(* IEC 61131-3 sources: plc-home-automation/home_automation/lighting_heating_updated/src/ventillation, 4 files *)

(* ---- VentillationGlobals.st ---- *)
VAR_GLOBAL CONSTANT

  C_NILAN_READ_COMMAND_GROUP : USINT          := 01;
  C_NILAN_SET_VENTILLATION_LEVEL_COMMAND_GROUP : USINT  := 02;
  C_NILAN_SET_DESIRED_TEMPERATURE_COMMAND_GROUP : USINT := 03;

  C_NUMBER_OF_NILAN_COMMANDS : USINT := 8;

  C_NILAN_STATUS_COMMAND_INDEX : USINT                    := 1;
  C_NILAN_STATUS_COMMAND_SIZE : UINT                        := 17;
  C_NILAN_ACTUAL_OPERATION_INDEX : USINT                  := 2;
  C_NILAN_ACTUAL_OPERATION_COMMAND_SIZE :UINT               := 4;
  C_NILAN_ACTUAL_VENTILLATION_INDEX : USINT               := 3;
  C_NILAN_ACTUAL_VENTILLATION_COMMAND_SIZE : UINT           := 5;
  C_CORE_DIAGNOSTICS_INDEX : USINT                        := 4;
  C_CORE_DIAGNOSTICS_COMMAND_SIZE : UINT                   := 23;
  C_CONTROLLED_TEMPERATURES_INDEX : USINT                 := 5;
  C_CONTROLLED_TEMPERATURES_COMMAND_SIZE : UINT             := 7;
  C_NILAN_SET_VENTILLATION_LEVEL_INDEX : USINT            := 6;
  C_NILAN_SET_VENTILLATION_LEVEL_COMMAND_SIZE : UINT        := 1;
  C_NILAN_SET_DESIRED_TEMPERATURE_INDEX : USINT           := 7;
  C_NILAN_SET_DESIRED_TEMPERATURE_COMMAND_SIZE : UINT       := 1;
  C_NILAN_ACTUAL_DISPLAY_GROUP_01_INDEX : UINT            := 8;
  C_NILAN_ACTUAL_DISPLAY_GROUP_01_COMMAND_SIZE : UINT       := 10;

  C_NILAN_MODBUS_ADDRESS : USINT := 30;

  C_NORMAL_VENTILLATION_LEVEL : INT := 1;
  C_BYPASS_VENTILLATION_LEVEL : INT := 3;

END_VAR

VAR_GLOBAL

  // User control
  PRESENCE_BASED_VENTILLATION_CONTROL   : BOOL := FALSE;
  COOLING_PRIORITY_VENTILLATION_CONTROL : BOOL := FALSE;

  // Read
  NILAN_COMMANDS : ARRAY [1..C_NUMBER_OF_NILAN_COMMANDS] OF TCmdStruct;

  NILAN_COMMAND_SIZES : ARRAY [1..C_NUMBER_OF_NILAN_COMMANDS] OF UINT;
  NILAN_COMMAND_BASE_ADRESSES : ARRAY [1..C_NUMBER_OF_NILAN_COMMANDS] OF UINT;
  NILAN_COMMAND_MODBUS_FNC : ARRAY [1..C_NUMBER_OF_NILAN_COMMANDS] OF USINT;
  NILAN_COMMAND_COMMAND_GROUP : ARRAY [1..C_NUMBER_OF_NILAN_COMMANDS] OF USINT;
  NILAN_COMMAND_DATA : ARRAY [1..C_NUMBER_OF_NILAN_COMMANDS] OF PTR_TO INT;

  NILAN_STATUS : ARRAY                    [1..C_NILAN_STATUS_COMMAND_SIZE] OF INT;
  NILAN_ACTUAL_OPERATION : ARRAY          [1..C_NILAN_ACTUAL_OPERATION_COMMAND_SIZE] OF INT;
  NILAN_ACTUAL_VENTILLATION : ARRAY       [1..C_NILAN_ACTUAL_VENTILLATION_COMMAND_SIZE] OF INT;
  NILAN_CORE_DIAGNOSTICS : ARRAY          [1..C_CORE_DIAGNOSTICS_COMMAND_SIZE] OF INT;
  NILAN_CONTROLLED_TEMPARATURES : ARRAY   [1..C_CONTROLLED_TEMPERATURES_COMMAND_SIZE] OF INT;
  NILAN_ACTUAL_DISPLAY_GROUP_01 : ARRAY   [1..C_NILAN_ACTUAL_DISPLAY_GROUP_01_COMMAND_SIZE] OF INT;

  NILAN_DESIRED_VENTILLATION_LEVEL : INT := 0;
  NILAN_DESIRED_TEMPERATURE        : INT := 24;
  NILAN_DESIRED_TEMPERATURE_SCALED : INT := 2400;

  // Alarms and warninrgs
  NILAN_ACTIVE_ERROR : BOOL := FALSE;
  NILAN_USER_FUNCTION : BOOL := FALSE;
  NILAN_AIR_FILTER_ALARM : BOOL := FALSE;

  // Ventillation
  NILAN_ACTUAL_VENTILLATION_SETPOINT          : INT := 0;
  NILAN_ACTUAL_VENTILLATION_INLET_FAN_LEVEL   : INT := 0;
  NILAN_ACTUAL_VENTILLATION_OUTLET_FAN_LEVEL  : INT := 0;
  NILAN_ACTUAL_VENTILLATION_AVERAGE_FAN_LEVEL : REAL := 0;

  // Core diagnostics (telemetry)
  NILAN_CONTROLLER_BOARD_TEMPERATURE : REAL := 0;

  NILAN_FRESH_AIR_INTAKE_TEMPERATURE    : REAL := 0;
  NILAN_INLET_TEMPERATURE_BEFORE_HEATER : REAL := 0;
  NILAN_ROOM_EXHAUST_TEMPERATURE        : REAL := 0;
  NILAN_OUTLET_TEMPERATURE              : REAL := 0;
  NILAN_CONDENSER_TEMPERATURE           : REAL := 0;
  NILAN_EVAPORATOR_TEMPERATURE          : REAL := 0;
  NILAN_INLET_TEMPERATURE_AFTER_HEATER  : REAL := 0;

  NILAN_OUTDOOR_TEMPERATURE : REAL := 0;

  NILAN_HEATING_SURFACE_TEMPERATURE : INT := 0;
  NILAN_EXTERNAL_ROOM_TEMPERATURE : INT := 0;
  NILAN_HOT_WATER_TOP_TEMPERATURE : INT := 0;
  NILAN_HOT_WATER_BOTTOM_TEMPERATURE : INT := 0;
  NILAN_EK_RETURN_TEMPERATURE : INT := 0;
  NILAN_EK_SUPPLY_TEMPERATURE : INT := 0;
  NILAN_USER_PANEL_ROOM_TEMPERATURE : INT := 0;
  NILAN_AUX_TEMPERATURE_HOTWATER_ANODE : INT := 0;
  NILAN_PREHEATER_OR_EARTH_TUBE_AIR_INTAKE_TEMPERATURE : INT := 0;
  NILAN_PRESSURE_PIBE_TEMPERATURE : INT := 0;
  NILAN_SUCTION_PRESSURE : INT := 0;
  NILAN_DISCHAGE_PRESSURE : INT := 0;
  NILAN_HUMIDITY_SENSOR_VALUE : REAL := 0;
  NILAN_CARBON_DIOXIDE_SENSOR_VALUE : INT := 0;
  NILAN_BYPASS_IS_ENABLED : BOOL := FALSE;

  // Furhter diagnostics
  NILAN_DAYS_SINCE_LAST_FILTER_CHANGE : INT := 0;
  NILAN_ACTUAL_CONTROLLED_TEMPERATURE : REAL := 0;

  NILAN_PASSIVE_HEAT_EXCHANGER_EFFICIENCY : REAL := 0;

END_VAR

(* ---- Ventillation.st ---- *)
PROGRAM VentillationControl

  VAR_INPUT
  END_VAR
  VAR_OUTPUT
  END_VAR
  VAR
     commUnit: fbModbusRTUmas2;
     modbusErrorMessage: String;

     presenceBasedDisable                 : BOOL := FALSE;
     coolingNeeded                        : BOOL := FALSE;

     setPresenceBasedVentillationToZero   : R_TRIG;
     setPresenceBasedVentillationToActive : F_TRIG;

     setCoolingBasedVentillationToZero    : F_TRIG;
     setCoolingBasedVentillationToActive  : R_TRIG;

     activateBypassVentialltionLevel      : R_TRIG;
     deactivateBypassVentialltionLevel    : F_TRIG;

     formerNilanDesiredVentillationLevel : INT := 0;
     formerNilanDesiredTemperature       : INT := 0;
     actualModbusCommandGroup            : USINT := C_NILAN_READ_COMMAND_GROUP;
  END_VAR
  VAR_TEMP
  END_VAR

  NILAN_DESIRED_TEMPERATURE_SCALED := NILAN_DESIRED_TEMPERATURE*100;

  coolingNeeded := (INT_TO_REAL(NILAN_DESIRED_TEMPERATURE) < NILAN_ACTUAL_CONTROLLED_TEMPERATURE) AND COOLING_PRIORITY_VENTILLATION_CONTROL;
  presenceBasedDisable := (GONE_FOR_5_HOURS OR (ALARM_ACTIVE AND GONE_FOR_5_HOURS)) AND NOT coolingNeeded AND PRESENCE_BASED_VENTILLATION_CONTROL;

  setPresenceBasedVentillationToZero(CLK := presenceBasedDisable);
  setPresenceBasedVentillationToACtive(CLK := presenceBasedDisable);

  setCoolingBasedVentillationToZero(CLK := coolingNeeded);
  setCoolingBasedVentillationToActive(CLK := coolingNeeded);

  activateBypassVentialltionLevel(CLK := NILAN_BYPASS_IS_ENABLED);
  deactivateBypassVentialltionLevel(CLK := NILAN_BYPASS_IS_ENABLED);

  // Turn off ventillation when no cooling is required and we're not at home
  IF setPresenceBasedVentillationToZero.Q THEN
    NILAN_DESIRED_VENTILLATION_LEVEL := 0;
  // Turn on ventillation someone is at home or we need cooling
  ELSIF setPresenceBasedVentillationToActive.Q OR setCoolingBasedVentillationToActive.Q THEN
    IF NILAN_BYPASS_IS_ENABLED THEN
      NILAN_DESIRED_VENTILLATION_LEVEL := C_BYPASS_VENTILLATION_LEVEL;
    ELSE
      NILAN_DESIRED_VENTILLATION_LEVEL := C_NORMAL_VENTILLATION_LEVEL;
    END_IF;
  END_IF;

  IF activateBypassVentialltionLevel.Q THEN
    IF NILAN_DESIRED_VENTILLATION_LEVEL < C_BYPASS_VENTILLATION_LEVEL THEN
      NILAN_DESIRED_VENTILLATION_LEVEL := C_BYPASS_VENTILLATION_LEVEL;
    END_IF;
  END_IF;

  IF deactivateBypassVentialltionLevel.Q THEN
    IF NILAN_DESIRED_VENTILLATION_LEVEL > C_NORMAL_VENTILLATION_LEVEL THEN
      NILAN_DESIRED_VENTILLATION_LEVEL := C_NORMAL_VENTILLATION_LEVEL;
    END_IF;
  END_IF;

  IF NOT formerNilanDesiredVentillationLevel = NILAN_DESIRED_VENTILLATION_LEVEL THEN

     actualModbusCommandGroup := C_NILAN_SET_VENTILLATION_LEVEL_COMMAND_GROUP;

     IF commUnit.LastCmd = C_NILAN_SET_VENTILLATION_LEVEL_INDEX THEN
       formerNilanDesiredVentillationLevel := NILAN_DESIRED_VENTILLATION_LEVEL;
     END_IF;

  ELSIF NOT formerNilanDesiredTemperature = NILAN_DESIRED_TEMPERATURE THEN

     actualModbusCommandGroup := C_NILAN_SET_DESIRED_TEMPERATURE_COMMAND_GROUP;

     IF commUnit.LastCmd = C_NILAN_SET_DESIRED_TEMPERATURE_INDEX THEN
       formerNilanDesiredTemperature := NILAN_DESIRED_TEMPERATURE;
     END_IF;

  ELSE

    actualModbusCommandGroup := C_NILAN_READ_COMMAND_GROUP;

  END_IF;

  commUnit(EN := true, GrSel := actualModbusCommandGroup, MaxCmd := C_NUMBER_OF_NILAN_COMMANDS,
             chanCode := CH2_uni, Endian := 0, Commands := NILAN_COMMANDS[1],
             MBtimeOut := T#30s, Delay := T#500ms);

  IF commUnit.ErrCode > 0 THEN
    GetModbusErrTxt(commUnit.ErrCode, modbusErrorMessage);
  END_IF;

  IF commUnit.Done THEN
     actualModbusCommandGroup := C_NILAN_READ_COMMAND_GROUP;
  END_IF;

  // Copy ventillation telemetry to global storage variables
  NILAN_USER_FUNCTION := INT_TO_BOOL(NILAN_STATUS[1]);
  NILAN_AIR_FILTER_ALARM := INT_TO_BOOL(NILAN_STATUS[2]);
  NILAN_ACTUAL_VENTILLATION_SETPOINT          := NILAN_ACTUAL_VENTILLATION[1];
  NILAN_ACTUAL_VENTILLATION_INLET_FAN_LEVEL   := NILAN_ACTUAL_VENTILLATION[2];
  NILAN_ACTUAL_VENTILLATION_OUTLET_FAN_LEVEL  := NILAN_ACTUAL_VENTILLATION[3];
  NILAN_ACTUAL_VENTILLATION_AVERAGE_FAN_LEVEL := INT_TO_REAL(NILAN_ACTUAL_VENTILLATION_INLET_FAN_LEVEL + NILAN_ACTUAL_VENTILLATION_OUTLET_FAN_LEVEL)/2;

  NILAN_CONTROLLER_BOARD_TEMPERATURE := INT_TO_REAL(NILAN_CORE_DIAGNOSTICS[1]) / 100;
  NILAN_FRESH_AIR_INTAKE_TEMPERATURE := INT_TO_REAL(NILAN_CORE_DIAGNOSTICS[2]) / 100;
  NILAN_INLET_TEMPERATURE_BEFORE_HEATER := INT_TO_REAL(NILAN_CORE_DIAGNOSTICS[3]) / 100;
  NILAN_ROOM_EXHAUST_TEMPERATURE := INT_TO_REAL(NILAN_CORE_DIAGNOSTICS[4]) / 100;
  NILAN_OUTLET_TEMPERATURE := INT_TO_REAL(NILAN_CORE_DIAGNOSTICS[5]) / 100;
  NILAN_CONDENSER_TEMPERATURE := INT_TO_REAL(NILAN_CORE_DIAGNOSTICS[6]) / 100;
  NILAN_EVAPORATOR_TEMPERATURE := INT_TO_REAL(NILAN_CORE_DIAGNOSTICS[7]) / 100;
  NILAN_INLET_TEMPERATURE_AFTER_HEATER := INT_TO_REAL(NILAN_CORE_DIAGNOSTICS[8]) / 100;
  NILAN_OUTDOOR_TEMPERATURE := INT_TO_REAL(NILAN_CORE_DIAGNOSTICS[9]) / 100;
  NILAN_HEATING_SURFACE_TEMPERATURE := NILAN_CORE_DIAGNOSTICS[10];
  NILAN_EXTERNAL_ROOM_TEMPERATURE := NILAN_CORE_DIAGNOSTICS[11];
  NILAN_HOT_WATER_TOP_TEMPERATURE := NILAN_CORE_DIAGNOSTICS[12];
  NILAN_HOT_WATER_BOTTOM_TEMPERATURE := NILAN_CORE_DIAGNOSTICS[13];
  NILAN_EK_RETURN_TEMPERATURE := NILAN_CORE_DIAGNOSTICS[14];
  NILAN_EK_SUPPLY_TEMPERATURE := NILAN_CORE_DIAGNOSTICS[15];
  NILAN_USER_PANEL_ROOM_TEMPERATURE := NILAN_CORE_DIAGNOSTICS[16];
  NILAN_AUX_TEMPERATURE_HOTWATER_ANODE := NILAN_CORE_DIAGNOSTICS[17];
  NILAN_PREHEATER_OR_EARTH_TUBE_AIR_INTAKE_TEMPERATURE := NILAN_CORE_DIAGNOSTICS[18];
  NILAN_PRESSURE_PIBE_TEMPERATURE := NILAN_CORE_DIAGNOSTICS[19];
  NILAN_SUCTION_PRESSURE := NILAN_CORE_DIAGNOSTICS[20];
  NILAN_DISCHAGE_PRESSURE := NILAN_CORE_DIAGNOSTICS[21];
  NILAN_HUMIDITY_SENSOR_VALUE := INT_TO_REAL(NILAN_CORE_DIAGNOSTICS[22])/100;
  NILAN_CARBON_DIOXIDE_SENSOR_VALUE := NILAN_CORE_DIAGNOSTICS[23];

  NILAN_DAYS_SINCE_LAST_FILTER_CHANGE := NILAN_ACTUAL_DISPLAY_GROUP_01[7];
  NILAN_BYPASS_IS_ENABLED := INT_TO_BOOL(NILAN_ACTUAL_DISPLAY_GROUP_01[1]);

  NILAN_ACTUAL_CONTROLLED_TEMPERATURE := INT_TO_REAL(NILAN_CONTROLLED_TEMPARATURES[3])/100;

  // This should by scaled by 100 according to the docs, but then I have 100%+ efficiency
  NILAN_PASSIVE_HEAT_EXCHANGER_EFFICIENCY := INT_TO_REAL(NILAN_CONTROLLED_TEMPARATURES[5])/100;

  // Flagging errors requiring physical attention
  NILAN_ACTIVE_ERROR := FALSE;

  IF NILAN_USER_FUNCTION THEN
    NILAN_ACTIVE_ERROR := TRUE;
  END_IF;

END_PROGRAM

(* ---- Ventillation_Control.st ---- *)
TYPE

  TemperatureDataBlock : STRUCT
    controllerBoardTemperature : REAL;
    IntakeTemperature : REAL;
    inletTemperature : REAL;
    exhaustTemparature : REAL;
    outletTemperature : REAL;
    condenserTemperature : REAL;
    evaporatorTemperature : REAL;
    afterHeatingInletTemperature : REAL;
    outdoorTemperature : REAL;
    heatingSurfaceTemperature : REAL;
END_STRUCT;

END_TYPE

VAR_GLOBAL CONSTANT
  C_NUMBER_OF_COMMANDS : SINT := 1;
END_VAR

VAR_GLOBAL
  Temps : TemperatureDataBlock;
  CmdCH2 : ARRAY [1..C_NUMBER_OF_COMMANDS] OF TCmdStruct;
END_VAR

PROGRAM Ventillation_Control

  VAR_INPUT
  END_VAR
  VAR_OUTPUT
  END_VAR
  VAR
     modbusUnit: ModbusRTUmas;
  END_VAR
  VAR_TEMP
  END_VAR

  ModbusCmd(Gr:=1, FNC:=03, SNo:=1,
  StAdr:=200, NoPoint:=SIZEOF(Temps)/2,
  PtrData:=adr(Temps), Cmd:=CmdCH2[1]);

  modbusUnit(EN := true, GrSel := 1, MaxCmd := C_NUMBER_OF_COMMANDS, chanCode := CH2_uni, Endian := 0, Commands := CmdCH2[1]);

END_PROGRAM

(* ---- VentillationInit.st ---- *)
PROGRAM VentillationInit
  VAR_INPUT
  END_VAR
  VAR_OUTPUT
  END_VAR
  VAR
    i : INT := 0;
    j : INT := 0;
    initialised : BOOL := FALSE;
  END_VAR
  VAR_TEMP
  END_VAR

  IF NOT initialised THEN

    NILAN_READ_COMMAND_SIZES[C_NILAN_STATUS_COMMAND_INDEX] :=       17;
    NILAN_READ_COMMAND_SIZES[C_NILAN_ACTUAL_OPERATION_INDEX] :=     4;
    NILAN_READ_COMMAND_SIZES[C_NILAN_ACTUAL_VENTILLATION_INDEX] :=  5;
    NILAN_READ_COMMAND_SIZES[C_CORE_TEMPERATURES_INDEX] :=          18;
    NILAN_READ_COMMAND_SIZES[C_CONTROLLED_TEMPERATURES_INDEX] :=    7;

    NILAN_READ_COMMAND_BASE_ADRESSES[C_NILAN_STATUS_COMMAND_INDEX] :=       100;
    NILAN_READ_COMMAND_BASE_ADRESSES[C_NILAN_ACTUAL_OPERATION_INDEX] :=     1000;
    NILAN_READ_COMMAND_BASE_ADRESSES[C_NILAN_ACTUAL_VENTILLATION_INDEX] :=  1100;
    NILAN_READ_COMMAND_BASE_ADRESSES[C_CORE_TEMPERATURES_INDEX] :=          200;
    NILAN_READ_COMMAND_BASE_ADRESSES[C_CONTROLLED_TEMPERATURES_INDEX] :=    1200;

    NILAN_READ_COMMAND_MODBUS_FNC[C_NILAN_STATUS_COMMAND_INDEX] :=       04;
    NILAN_READ_COMMAND_MODBUS_FNC[C_NILAN_ACTUAL_OPERATION_INDEX] :=     04;
    NILAN_READ_COMMAND_MODBUS_FNC[C_NILAN_ACTUAL_VENTILLATION_INDEX] :=  04;
    NILAN_READ_COMMAND_MODBUS_FNC[C_CORE_TEMPERATURES_INDEX] :=          04;
    NILAN_READ_COMMAND_MODBUS_FNC[C_CONTROLLED_TEMPERATURES_INDEX] :=    04;

    NILAN_VENTILLATION_SET_FAN_LEVEL_COMMAND_SIZES[C_NILAN_STATUS_COMMAND_INDEX] :=         1;

    NILAN_VENTILLATION_SET_FAN_LEVEL_COMMAND_BASE_ADRESSES[C_NILAN_STATUS_COMMAND_INDEX] := 1003;

    NILAN_VENTILLATION_SET_FAN_LEVEL_COMMAND_MODBUS_FNC[C_NILAN_STATUS_COMMAND_INDEX] :=    16;

    FOR i := 0 TO C_NUMBER_OF_NILAN_COMMAND_GROUPS DO
      FOR j := 0 TO NUMBER_OF_COMMANDS_IN_NILAN_COMMAND_GROUP[i] DO
         NILAN_COMMAND_BASE_ADDRESS

         ModbusCmd(Gr:=i, FNC:=NILAN_COMMAND_FNC + j*size, SNo:=C_NILAN_MODBUS_ADDRESS,
          StAdr:=C_NILAN_STATUS_BASE_ADDRESS, NoPoint:=C_NILAN_STATUS_SIZE,
          PtrData:=adr(NILAN_STATUS), Cmd:=VENTILLATION_READ_COMMANDS[1])
      END_FOR;
    END_FOR;

    ModbusCmd(Gr:=1, FNC:=C_NILAN_STATUS_MODBUS_FNC, SNo:=C_NILAN_MODBUS_ADDRESS,
    StAdr:=C_NILAN_STATUS_BASE_ADDRESS, NoPoint:=C_NILAN_STATUS_SIZE,
    PtrData:=adr(NILAN_STATUS), Cmd:=VENTILLATION_READ_COMMANDS[1]);

    ModbusCmd(Gr:=1, FNC:=C_NILAN_ACTUAL_OPERATION_MODBUS_FNC, SNo:=C_NILAN_MODBUS_ADDRESS,
    StAdr:=C_NILAN_ACTUAL_OPERATION_BASE_ADDRESS, NoPoint:=C_NILAN_ACTUAL_OPERATION_SIZE,
    PtrData:=adr(NILAN_ACTUAL_OPERATION), Cmd:=VENTILLATION_READ_COMMANDS[2]);

    ModbusCmd(Gr:=1, FNC:=C_NILAN_ACTUAL_VENTILLATION_MODBUS_FNC, SNo:=C_NILAN_MODBUS_ADDRESS,
    StAdr:=C_NILAN_ACTUAL_VENTILLATION_BASE_ADDRESS, NoPoint:=C_NILAN_ACTUAL_VENTILLATION_SIZE,
    PtrData:=adr(NILAN_ACTUAL_VENTILLATION), Cmd:=VENTILLATION_READ_COMMANDS[3]);

    ModbusCmd(Gr:=1, FNC:=C_CORE_TEMPERATURES_MODBUS_FNC, SNo:=C_NILAN_MODBUS_ADDRESS,
    StAdr:=C_CORE_TEMPERATURES_BASE_ADDRESS, NoPoint:=C_CORE_TEMPERATURES_SIZE,
    PtrData:=adr(CORE_TEMPARATURES), Cmd:=VENTILLATION_READ_COMMANDS[4]);

    ModbusCmd(Gr:=1, FNC:=C_CONTROLLED_TEMPERATURES_MODBUS_FNC, SNo:=C_NILAN_MODBUS_ADDRESS,
    StAdr:=C_CONTROLLED_TEMPERATURES_BASE_ADDRESS, NoPoint:=C_CONTROLLED_TEMPERATURES_SIZE,
    PtrData:=adr(CONTROLLED_TEMPARATURES), Cmd:=VENTILLATION_READ_COMMANDS[5]);

    ModbusCmd(Gr:=1, FNC:=C_VENTILLATION_SET_FAN_LEVEL_MODBUS_FNC, SNo:=C_NILAN_MODBUS_ADDRESS,
    StAdr:=C_VENTILLATION_SET_FAN_LEVEL_BASE_ADDRESS, NoPoint:=C_VENTILLATION_SET_FAN_LEVEL_SIZE,
    PtrData:=adr(DESIRED_VENTILLATION_LEVEL), Cmd:=VENTILLATION_SET_FAN_LEVEL_COMMAND[1]);

    initialised := TRUE;
  END_IF

END_PROGRAM
